FUNCTION_BLOCK FB_TextFile
VAR_INPUT
END_VAR
VAR_OUTPUT
END_VAR
VAR
END_VAR

METHOD Read : BOOL
VAR_INPUT
END_VAR
END_METHOD

END_FUNCTION_BLOCK

(* stored: Version 1.1.0.1
   POU FB_TextFile: Id {a8fbbdb2-8622-4f28-96c1-2e6d5da1b20c}, SpecialFunc None
   Method Read: Id {125b370c-fee2-4bc3-952c-f17051a924a3} *)
